// SIMATIC S7-200 project (STEP 7-Micro/WIN), CPU 224XP REL 02.01

ORGANIZATION_BLOCK 程序块:OB1
TITLE=程序注释
BEGIN
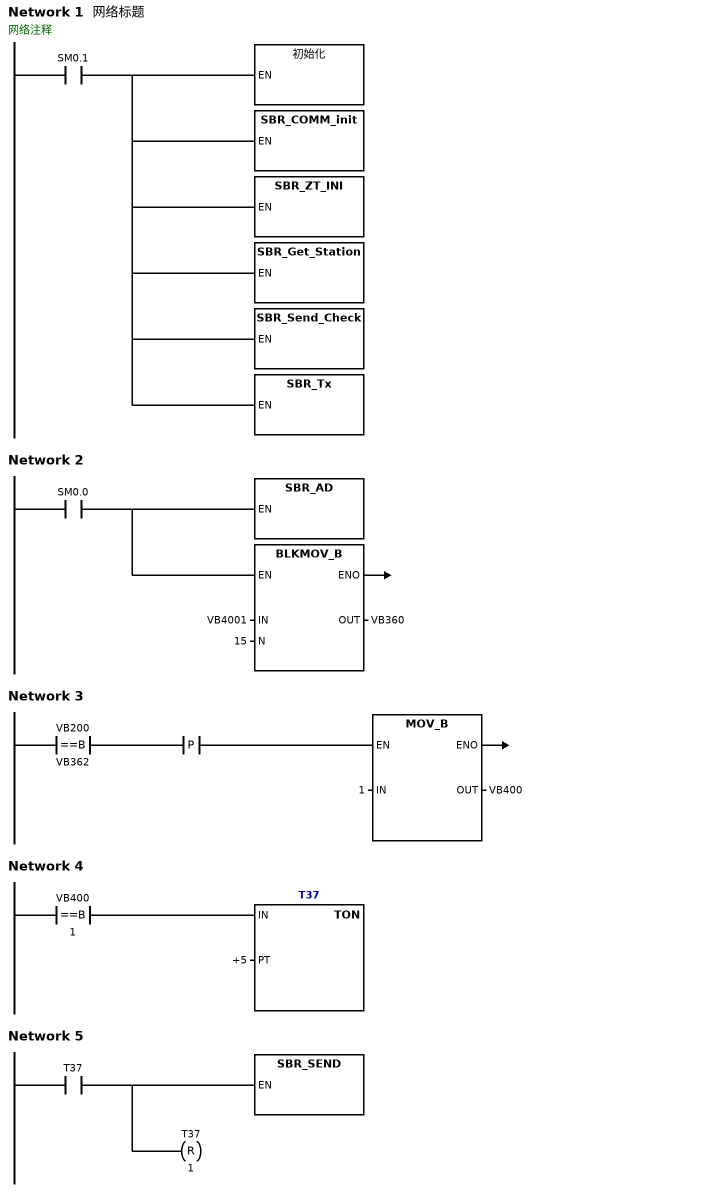
Network 1 // 网络标题
// 网络注释
LD     SM0.1
CALL   初始化:SBR0
CALL   SBR_COMM_init:SBR1
CALL   SBR_ZT_INI:SBR11
CALL   SBR_Get_Station:SBR15
CALL   SBR_Send_Check:SBR14
CALL   SBR_Tx:SBR17
Network 2
LD     SM0.0
CALL   SBR_AD:SBR19
BMB    VB4001, VB360, 15
Network 3
LDB=   VB200, VB362
EU
MOVB   1, VB400
Network 4
LDB=   VB400, 1
TON    T37, +5
Network 5
LD     T37
CALL   SBR_SEND:SBR9
R      T37, 1
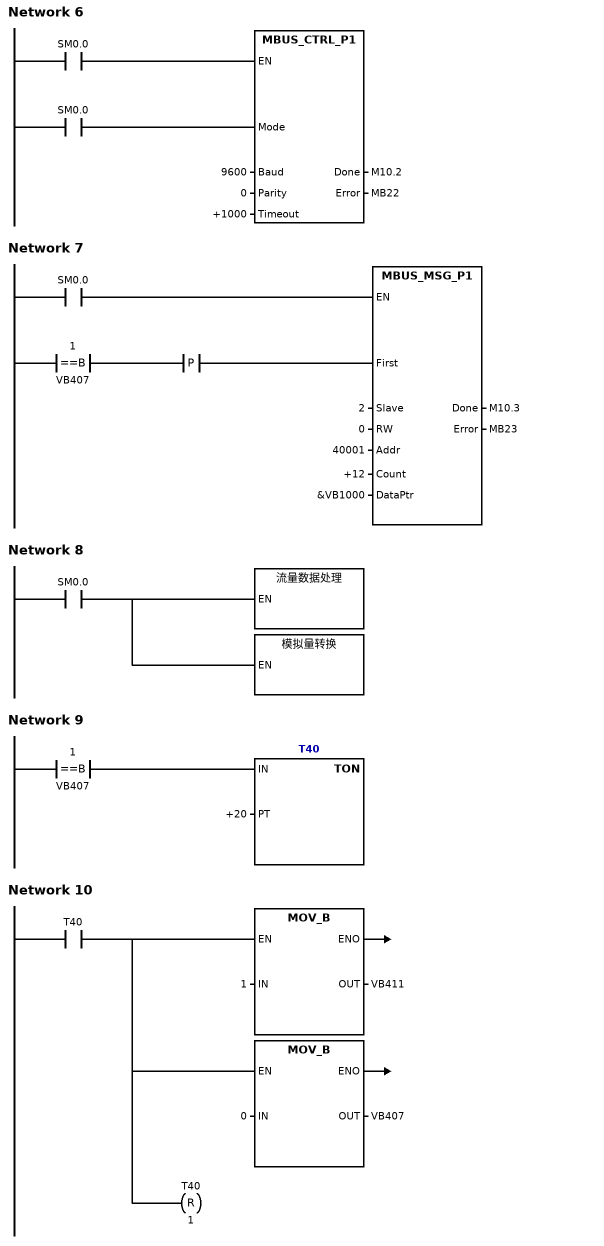
Network 6
LD     SM0.0
=      L60.0
LD     SM0.0
=      L63.7
LD     L60.0
CALL   MBUS_CTRL_P1:SBR6, L63.7, 9600, 0, +1000, M10.2, MB22
Network 7
LD     SM0.0
=      L60.0
LDB=   1, VB407
EU
=      L63.7
LD     L60.0
CALL   MBUS_MSG_P1:SBR7, L63.7, 2, 0, 40001, +12, &VB1000, M10.3, MB23
Network 8
LD     SM0.0
CALL   流量数据处理:SBR2
CALL   模拟量转换:SBR10
Network 9
LDB=   1, VB407
TON    T40, +20
Network 10
LD     T40
MOVB   1, VB411
MOVB   0, VB407
R      T40, 1
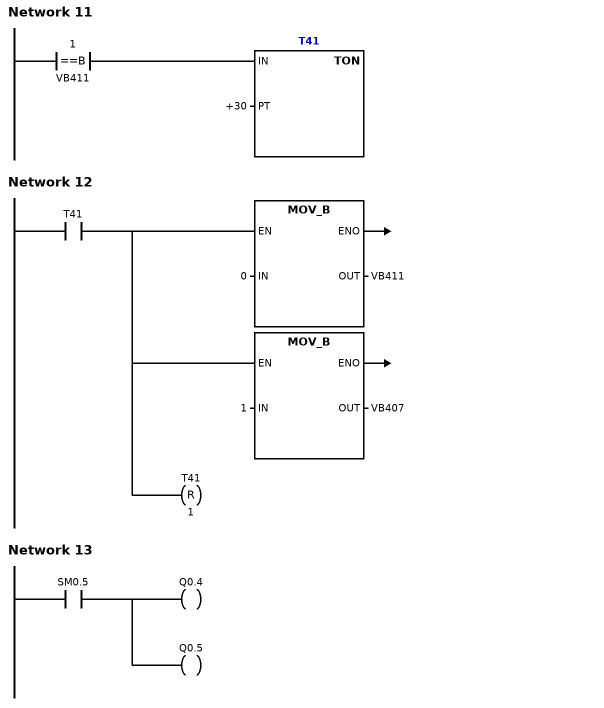
Network 11
LDB=   1, VB411
TON    T41, +30
Network 12
LD     T41
MOVB   0, VB411
MOVB   1, VB407
R      T41, 1
Network 13
LD     SM0.5
=      Q0.4
=      Q0.5
END_ORGANIZATION_BLOCK

SUBROUTINE_BLOCK 初始化:SBR0
TITLE=子程序注释
BEGIN
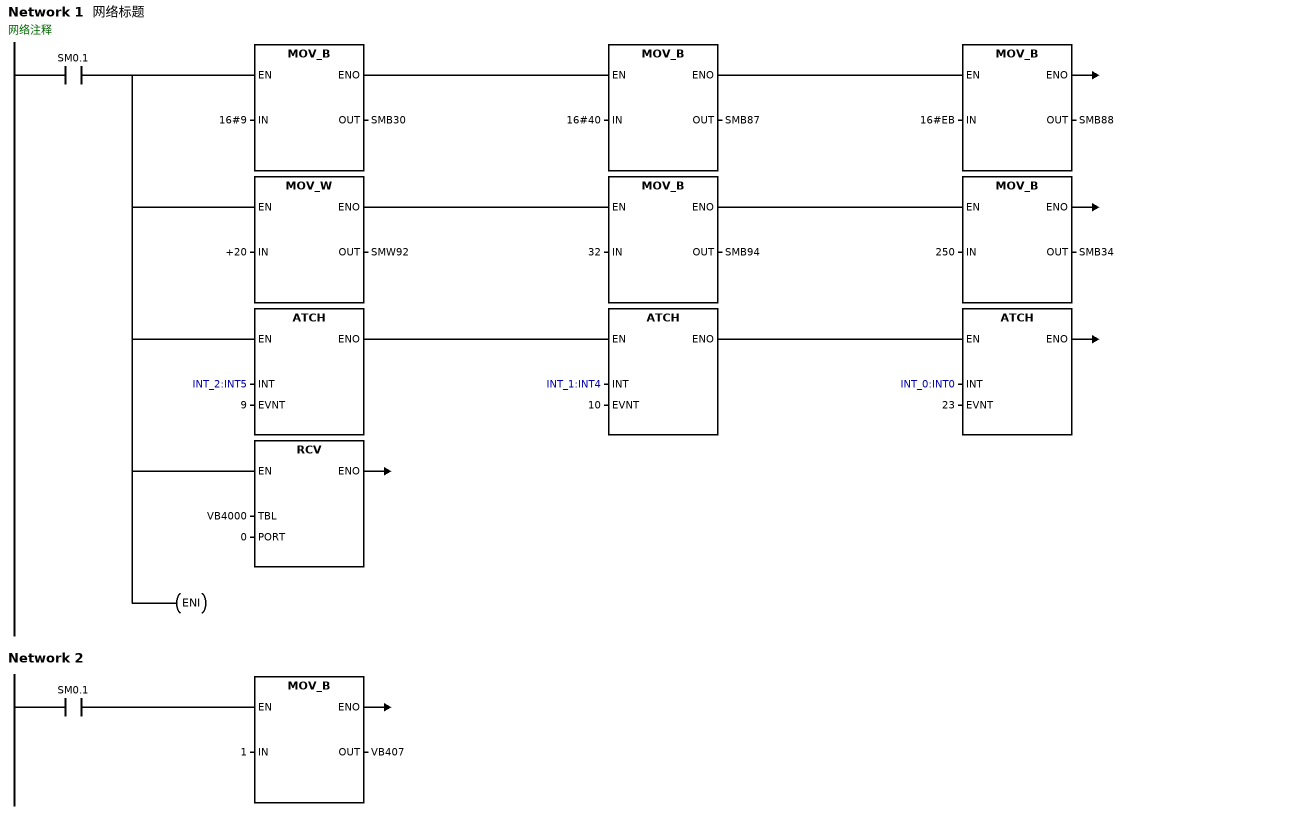
Network 1 // 网络标题
// 网络注释
LD     SM0.1
LPS
MOVB   16#9, SMB30
AENO
MOVB   16#40, SMB87
AENO
MOVB   16#EB, SMB88
LRD
MOVW   +20, SMW92
AENO
MOVB   32, SMB94
AENO
MOVB   250, SMB34
LRD
ATCH   INT_2:INT5, 9
AENO
ATCH   INT_1:INT4, 10
AENO
ATCH   INT_0:INT0, 23
LRD
RCV    VB4000, 0
LPP
ENI
Network 2
LD     SM0.1
MOVB   1, VB407
END_SUBROUTINE_BLOCK

SUBROUTINE_BLOCK SBR_COMM_init:SBR1
TITLE=
BEGIN
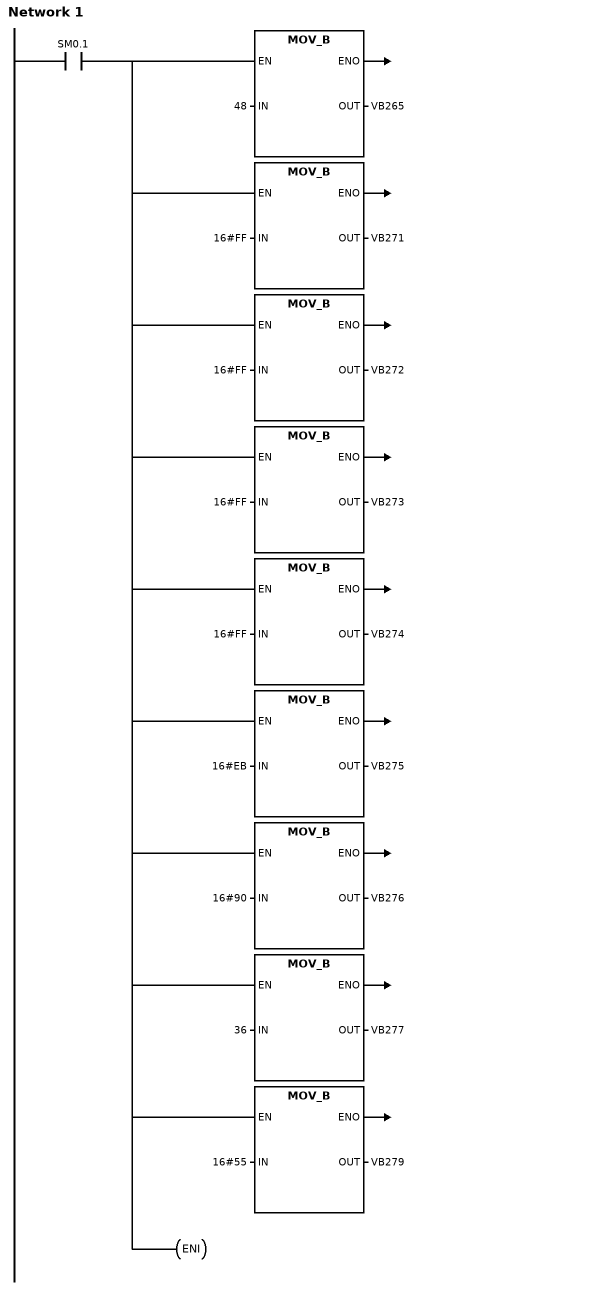
Network 1
LD     SM0.1
MOVB   48, VB265
MOVB   16#FF, VB271
MOVB   16#FF, VB272
MOVB   16#FF, VB273
MOVB   16#FF, VB274
MOVB   16#EB, VB275
MOVB   16#90, VB276
MOVB   36, VB277
MOVB   16#55, VB279
ENI
END_SUBROUTINE_BLOCK

SUBROUTINE_BLOCK 流量数据处理:SBR2
TITLE=
BEGIN
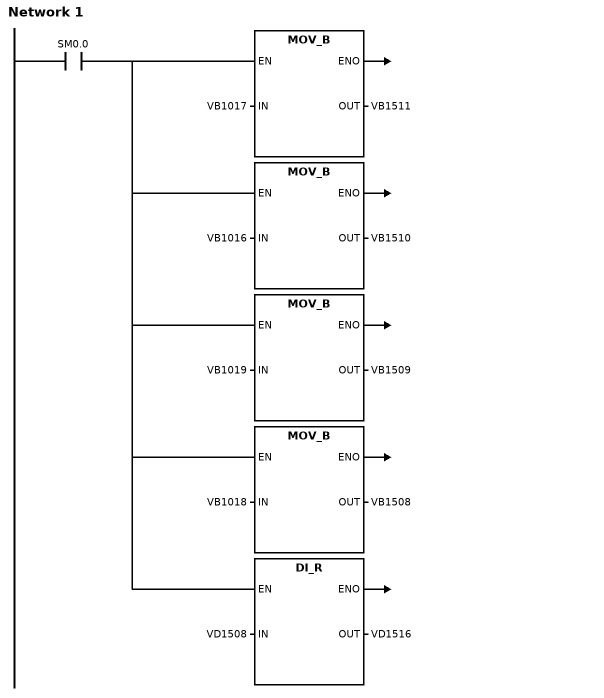
Network 1
LD     SM0.0
MOVB   VB1017, VB1511
MOVB   VB1016, VB1510
MOVB   VB1019, VB1509
MOVB   VB1018, VB1508
DTR    VD1508, VD1516
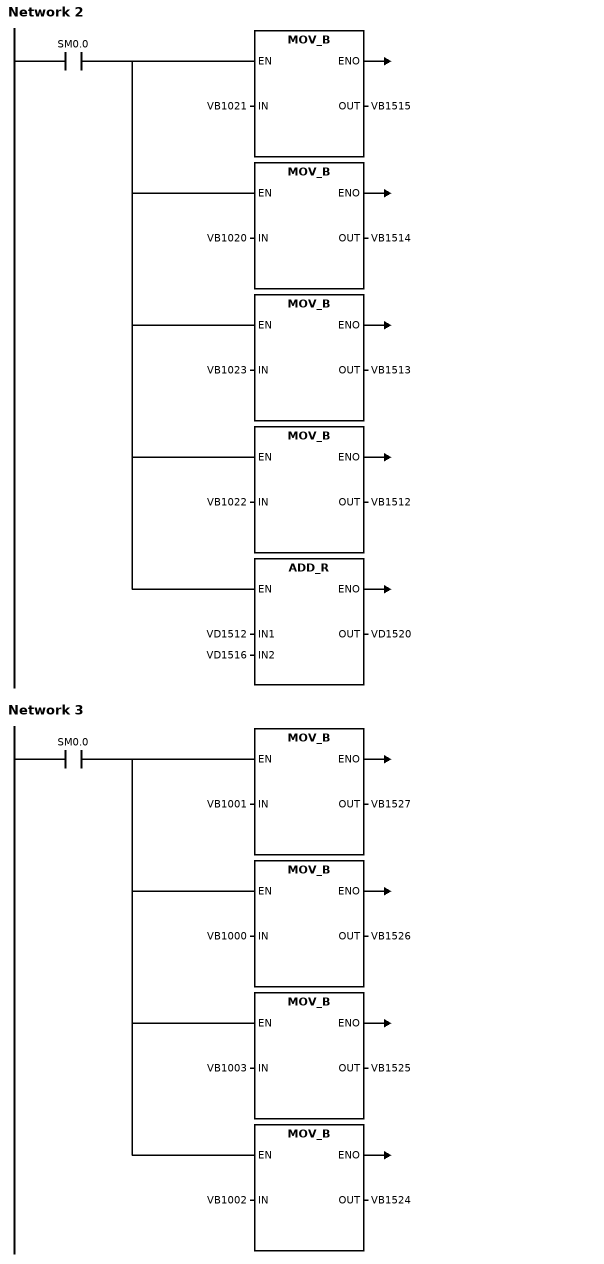
Network 2
LD     SM0.0
MOVB   VB1021, VB1515
MOVB   VB1020, VB1514
MOVB   VB1023, VB1513
MOVB   VB1022, VB1512
MOVR   VD1512, VD1520
+R     VD1516, VD1520
Network 3
LD     SM0.0
MOVB   VB1001, VB1527
MOVB   VB1000, VB1526
MOVB   VB1003, VB1525
MOVB   VB1002, VB1524
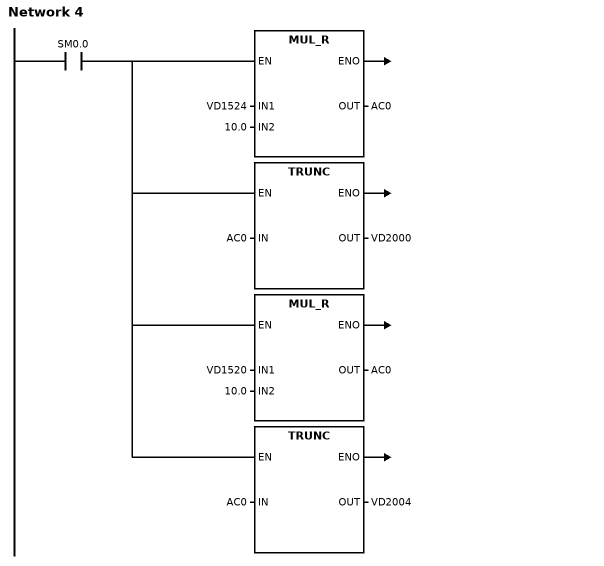
Network 4
LD     SM0.0
MOVR   VD1524, AC0
*R     10.0, AC0
TRUNC  AC0, VD2000
MOVR   VD1520, AC0
*R     10.0, AC0
TRUNC  AC0, VD2004
END_SUBROUTINE_BLOCK

// SBR3: protected block, not included

// SBR4: protected block, not included

// SBR5: protected block, not included

// SBR6: protected block, not included

// SBR7: protected block, not included

// SBR8: protected block, not included

SUBROUTINE_BLOCK SBR_SEND:SBR9
TITLE=
BEGIN
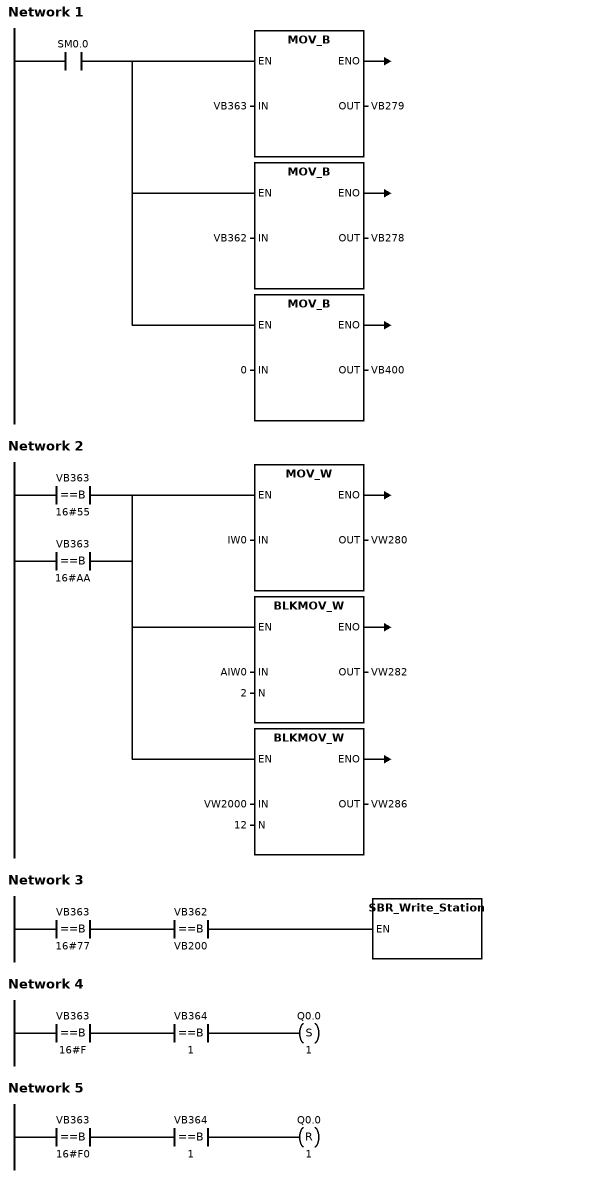
Network 1
LD     SM0.0
MOVB   VB363, VB279
MOVB   VB362, VB278
MOVB   0, VB400
Network 2
LDB=   VB363, 16#55
OB=    VB363, 16#AA
MOVW   IW0, VW280
BMW    AIW0, VW282, 2
BMW    VW2000, VW286, 12
Network 3
LDB=   VB363, 16#77
AB=    VB362, VB200
CALL   SBR_Write_Station:SBR16
Network 4
LDB=   VB363, 16#F
AB=    VB364, 1
S      Q0.0, 1
Network 5
LDB=   VB363, 16#F0
AB=    VB364, 1
R      Q0.0, 1
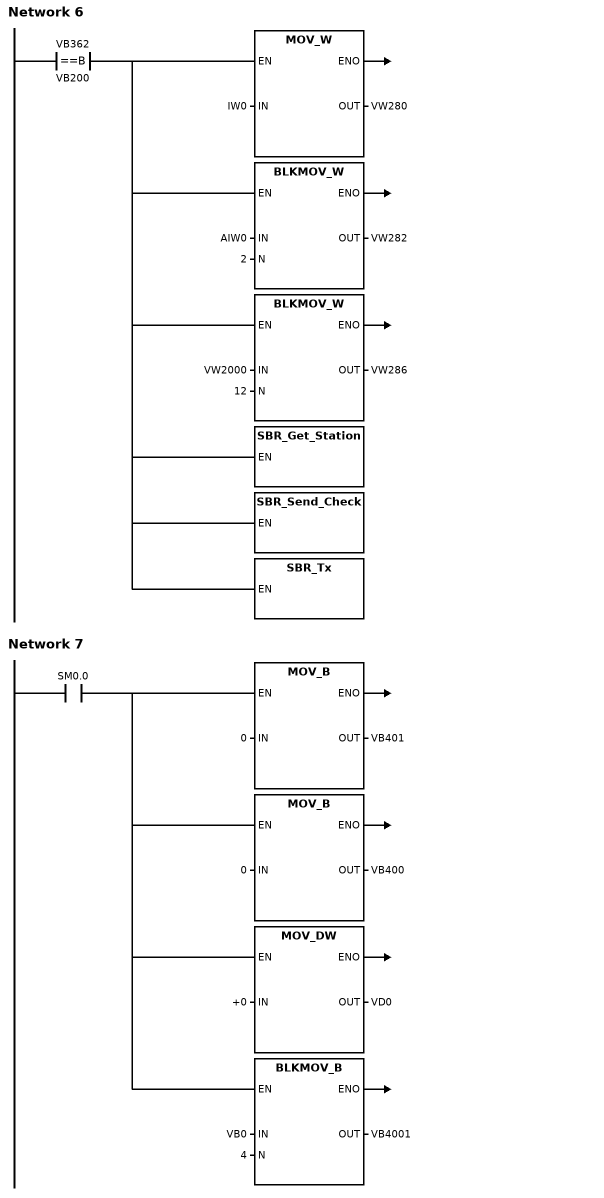
Network 6
LDB=   VB362, VB200
MOVW   IW0, VW280
BMW    AIW0, VW282, 2
BMW    VW2000, VW286, 12
CALL   SBR_Get_Station:SBR15
CALL   SBR_Send_Check:SBR14
CALL   SBR_Tx:SBR17
Network 7
LD     SM0.0
MOVB   0, VB401
MOVB   0, VB400
MOVD   +0, VD0
BMB    VB0, VB4001, 4
END_SUBROUTINE_BLOCK

SUBROUTINE_BLOCK 模拟量转换:SBR10
TITLE=
BEGIN
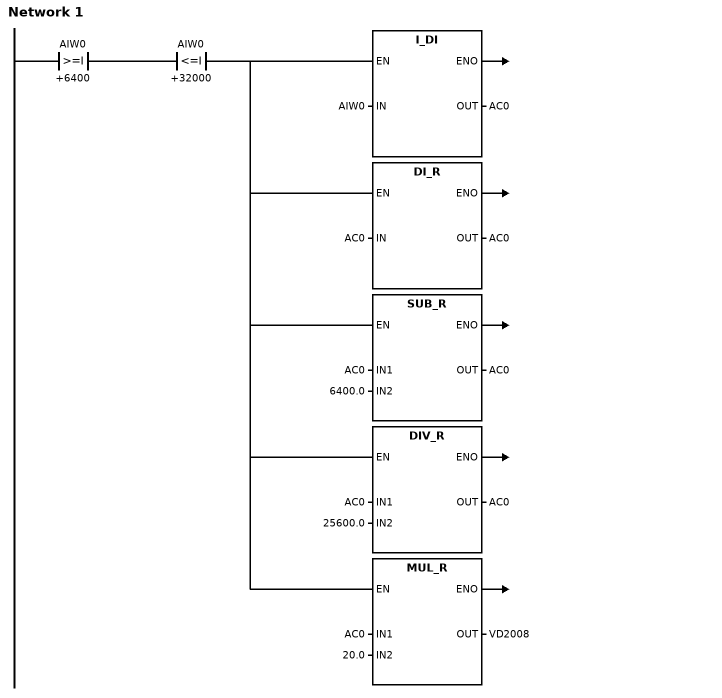
Network 1
LDW>=  AIW0, +6400
AW<=   AIW0, +32000
ITD    AIW0, AC0
DTR    AC0, AC0
-R     6400.0, AC0
/R     25600.0, AC0
MOVR   AC0, VD2008
*R     20.0, VD2008
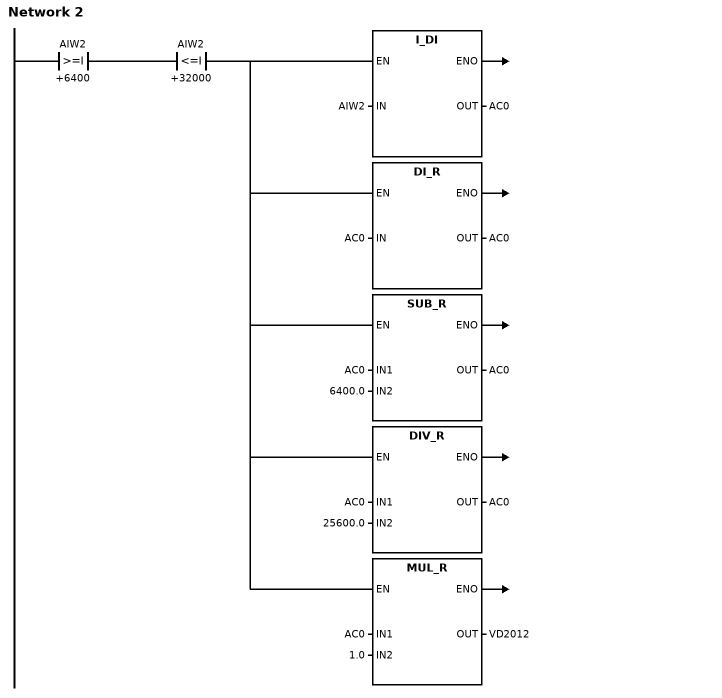
Network 2
LDW>=  AIW2, +6400
AW<=   AIW2, +32000
ITD    AIW2, AC0
DTR    AC0, AC0
-R     6400.0, AC0
/R     25600.0, AC0
MOVR   AC0, VD2012
*R     1.0, VD2012
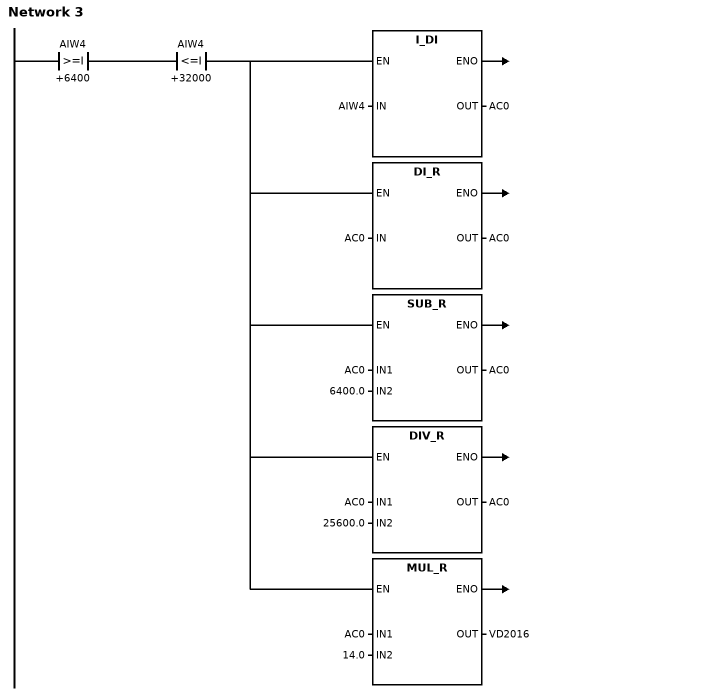
Network 3
LDW>=  AIW4, +6400
AW<=   AIW4, +32000
ITD    AIW4, AC0
DTR    AC0, AC0
-R     6400.0, AC0
/R     25600.0, AC0
MOVR   AC0, VD2016
*R     14.0, VD2016
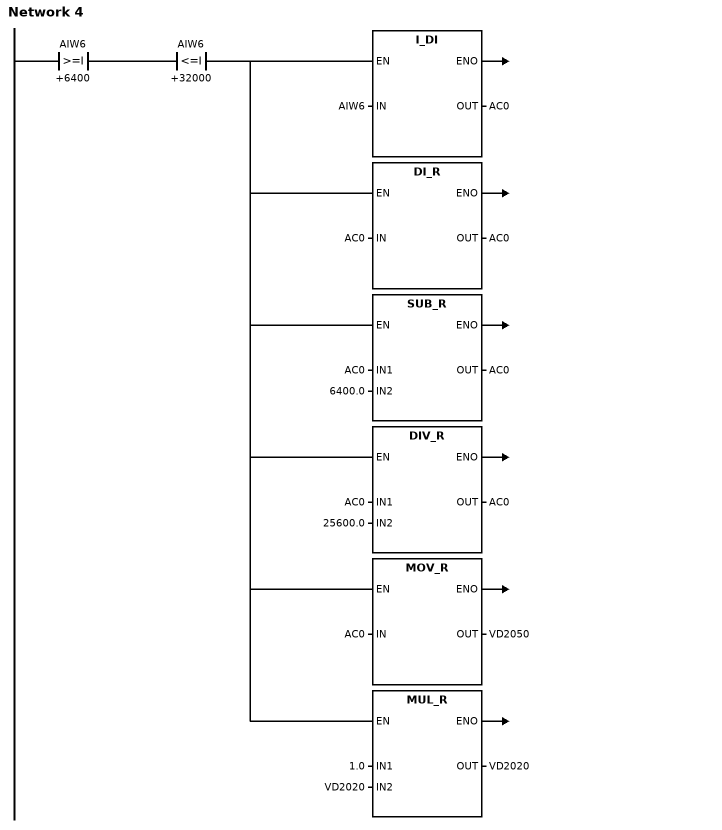
Network 4
LDW>=  AIW6, +6400
AW<=   AIW6, +32000
ITD    AIW6, AC0
DTR    AC0, AC0
-R     6400.0, AC0
/R     25600.0, AC0
MOVR   AC0, VD2050
*R     1.0, VD2020
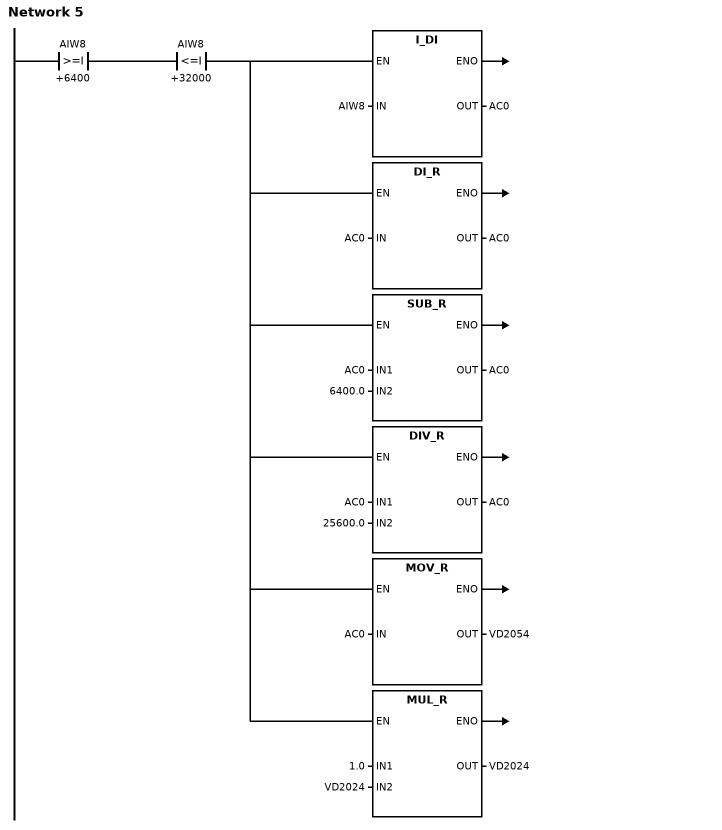
Network 5
LDW>=  AIW8, +6400
AW<=   AIW8, +32000
ITD    AIW8, AC0
DTR    AC0, AC0
-R     6400.0, AC0
/R     25600.0, AC0
MOVR   AC0, VD2054
*R     1.0, VD2024
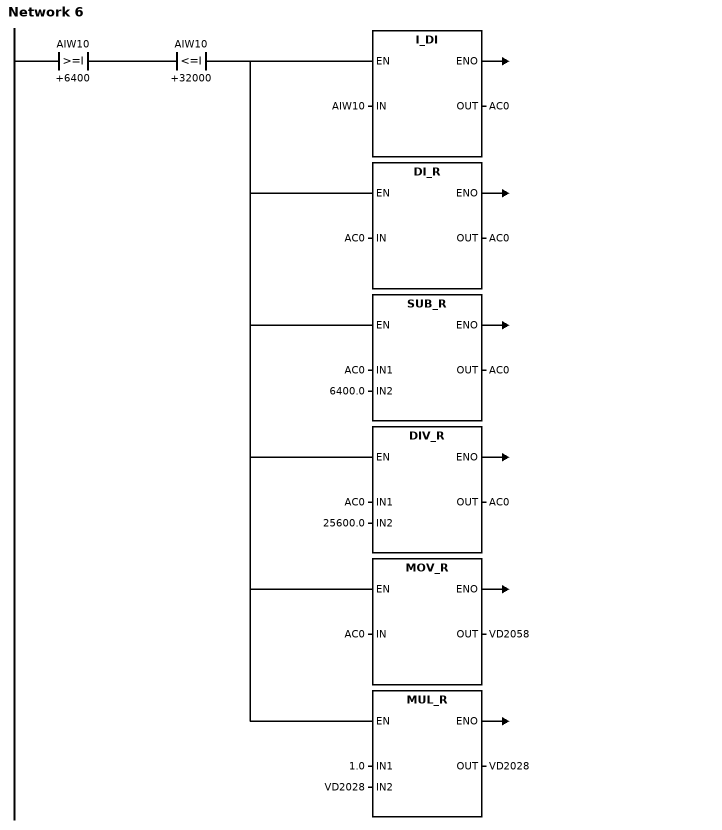
Network 6
LDW>=  AIW10, +6400
AW<=   AIW10, +32000
ITD    AIW10, AC0
DTR    AC0, AC0
-R     6400.0, AC0
/R     25600.0, AC0
MOVR   AC0, VD2058
*R     1.0, VD2028
END_SUBROUTINE_BLOCK

SUBROUTINE_BLOCK SBR_ZT_INI:SBR11
TITLE=
BEGIN
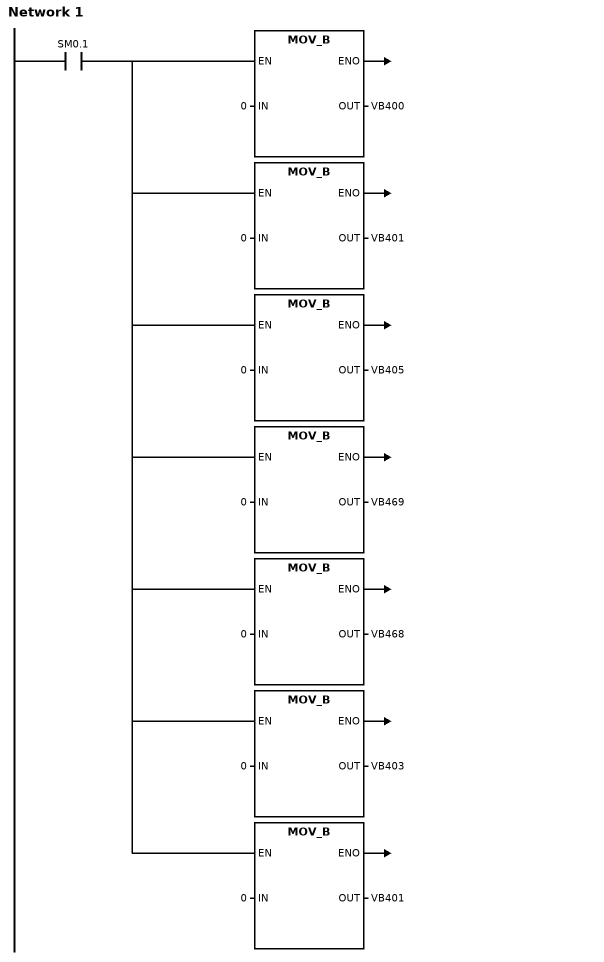
Network 1
LD     SM0.1
MOVB   0, VB400
MOVB   0, VB401
MOVB   0, VB405
MOVB   0, VB469
MOVB   0, VB468
MOVB   0, VB403
MOVB   0, VB401
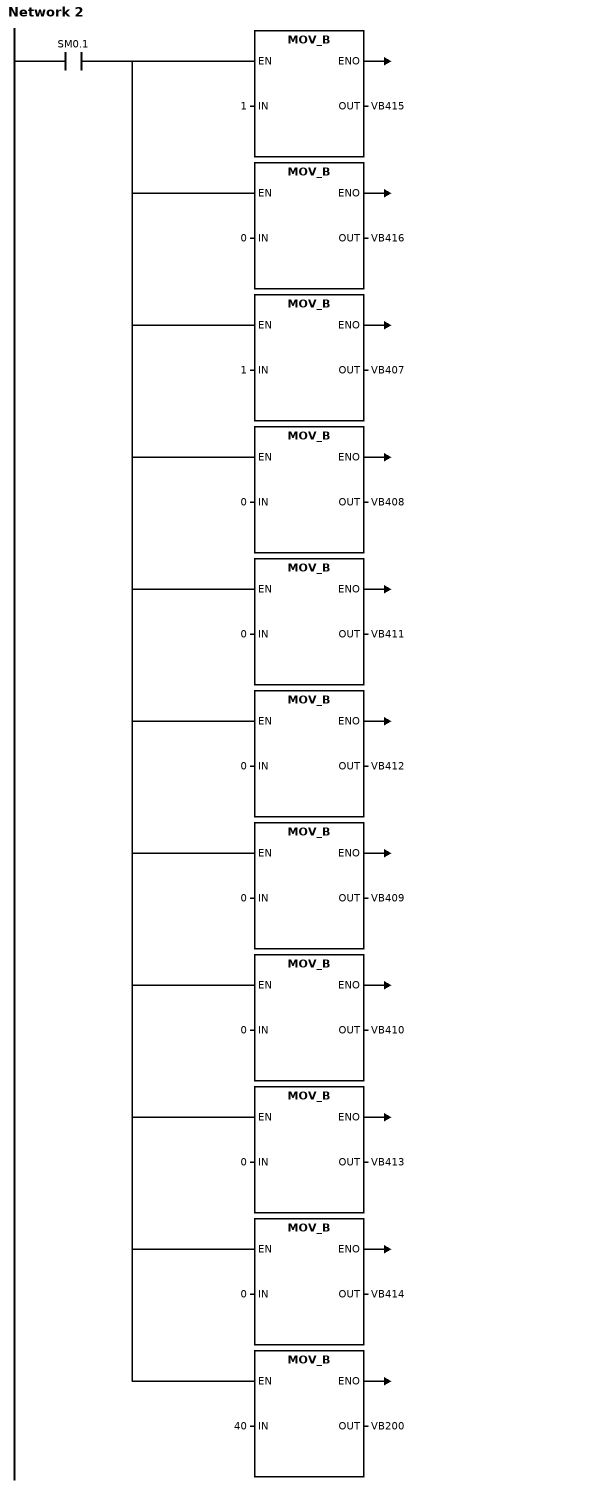
Network 2
LD     SM0.1
MOVB   1, VB415
MOVB   0, VB416
MOVB   1, VB407
MOVB   0, VB408
MOVB   0, VB411
MOVB   0, VB412
MOVB   0, VB409
MOVB   0, VB410
MOVB   0, VB413
MOVB   0, VB414
MOVB   40, VB200
END_SUBROUTINE_BLOCK

SUBROUTINE_BLOCK SBR_Jscl:SBR12
TITLE=
BEGIN
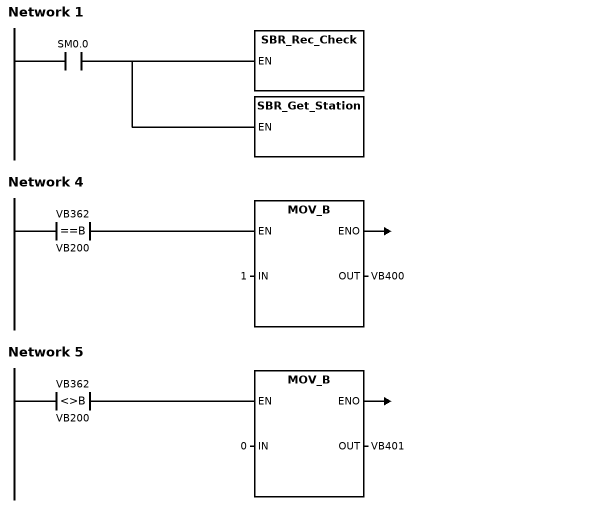
Network 1
LD     SM0.0
CALL   SBR_Rec_Check:SBR13
CALL   SBR_Get_Station:SBR15
Network 4
LDB=   VB362, VB200
MOVB   1, VB400
Network 5
LDB<>  VB362, VB200
MOVB   0, VB401
END_SUBROUTINE_BLOCK

SUBROUTINE_BLOCK SBR_Rec_Check:SBR13
TITLE=
BEGIN
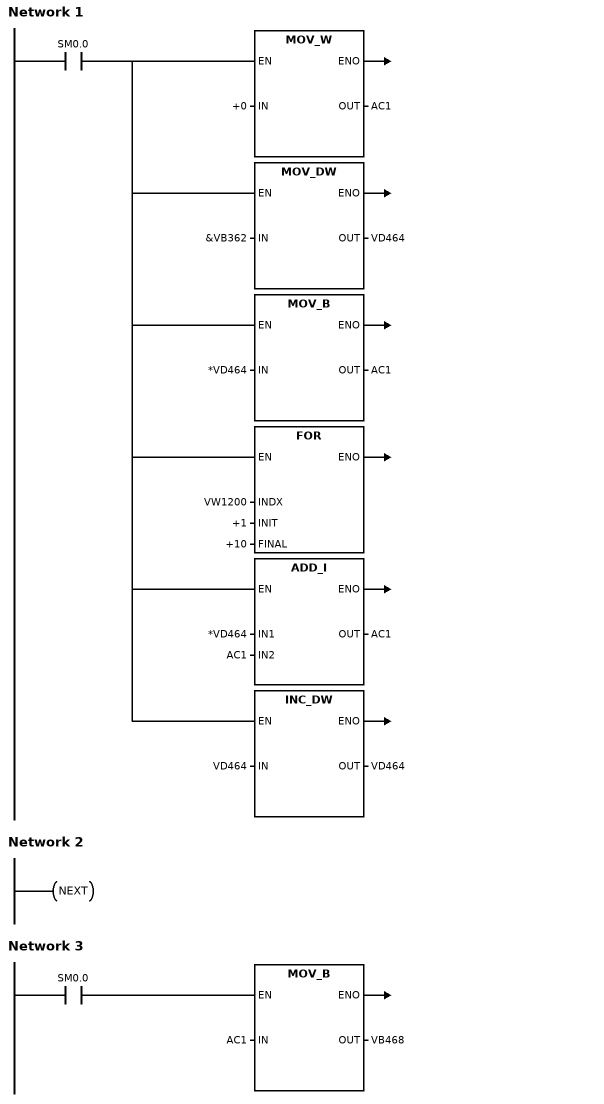
Network 1
LD     SM0.0
MOVW   +0, AC1
MOVD   &VB362, VD464
MOVB   *VD464, AC1
FOR    VW1200, +1, +10
+I     *VD464, AC1
INCD   VD464
Network 2
NEXT
Network 3
LD     SM0.0
MOVB   AC1, VB468
END_SUBROUTINE_BLOCK

SUBROUTINE_BLOCK SBR_Send_Check:SBR14
TITLE=
BEGIN
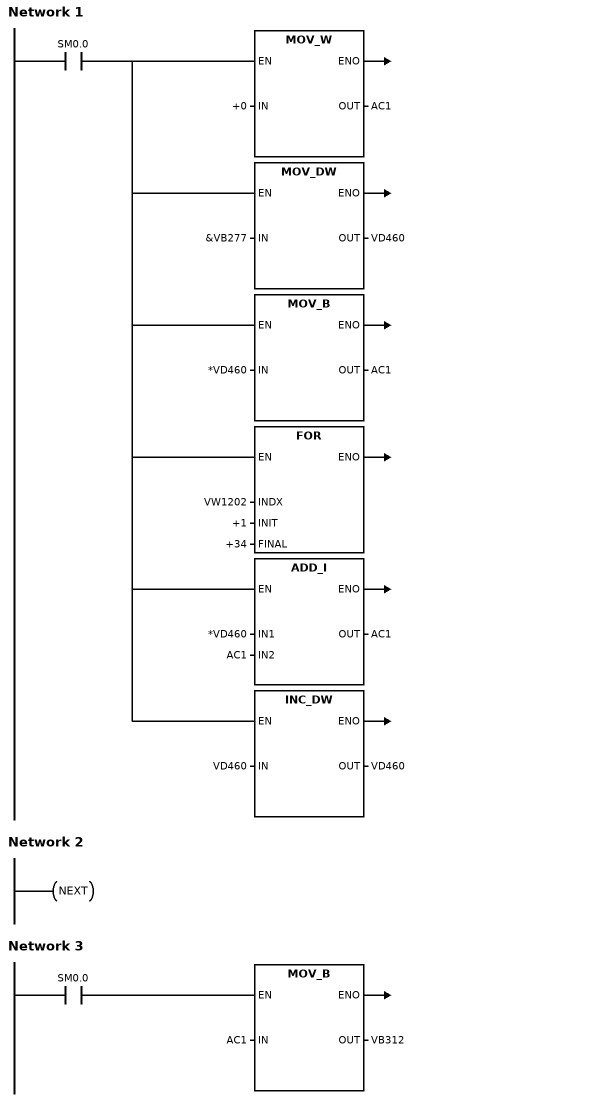
Network 1
LD     SM0.0
MOVW   +0, AC1
MOVD   &VB277, VD460
MOVB   *VD460, AC1
FOR    VW1202, +1, +34
+I     *VD460, AC1
INCD   VD460
Network 2
NEXT
Network 3
LD     SM0.0
MOVB   AC1, VB312
END_SUBROUTINE_BLOCK

SUBROUTINE_BLOCK SBR_Get_Station:SBR15
TITLE=
BEGIN
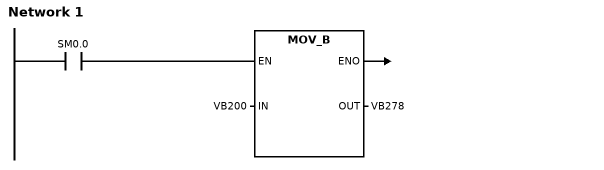
Network 1
LD     SM0.0
MOVB   VB200, VB278
END_SUBROUTINE_BLOCK

SUBROUTINE_BLOCK SBR_Write_Station:SBR16
TITLE=
BEGIN
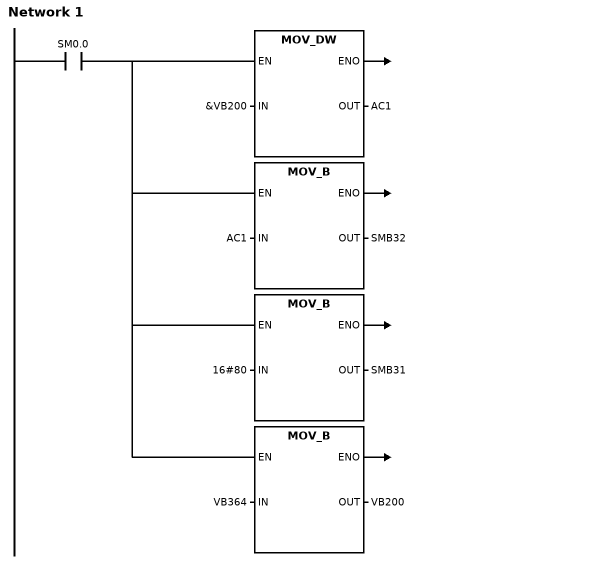
Network 1
LD     SM0.0
MOVD   &VB200, AC1
MOVB   AC1, SMB32
MOVB   16#80, SMB31
MOVB   VB364, VB200
END_SUBROUTINE_BLOCK

SUBROUTINE_BLOCK SBR_Tx:SBR17
TITLE=
BEGIN
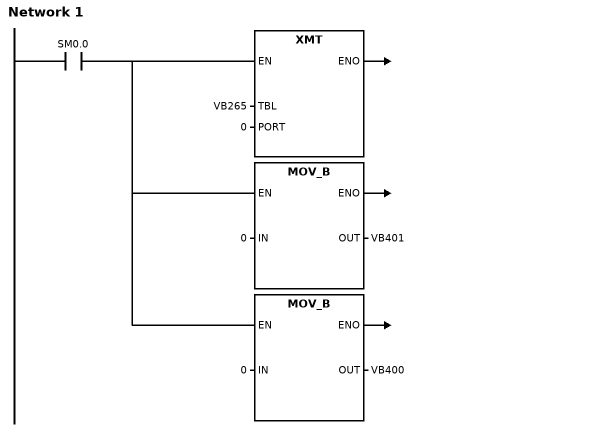
Network 1
LD     SM0.0
XMT    VB265, 0
MOVB   0, VB401
MOVB   0, VB400
END_SUBROUTINE_BLOCK

SUBROUTINE_BLOCK SBR_AD:SBR19
TITLE=
BEGIN
